// TIA Portal V17 export
// export: Created 2024-09-02T12:50:15.659418Z, ExportSetting WithDefaults, DisplayName Totally Integrated Automation Portal, DisplayVersion V17, DisplayName TIA Portal Openness, DisplayVersion V17, DisplayName TIA Portal Version Control Interface, DisplayVersion V17, DisplayName STEP 7 Professional, DisplayVersion V17, DisplayName STEP 7 Safety, DisplayVersion V17, DisplayName WinCC Professional, DisplayVersion V17
FUNCTION "AnwFC_ZP_InterfaceMainScreen_OP70" : Void   // FC163, LAD
TITLE = Station overview / Stationsübersicht
{ S7_Optimized_Access := 'TRUE' }
AUTHOR : OlegFuehrus
FAMILY : BA
NAME : BA
VERSION : 0.1
// stored: AutoNumber false, IsIECCheckEnabled false, SetENOAutomatically false, UDAEnableTagReadback false
   VAR_TEMP
      t_VKE0 : Bool;
      t_VKE1 : Bool;
   END_VAR
BEGIN

REGION Network 1: INIT
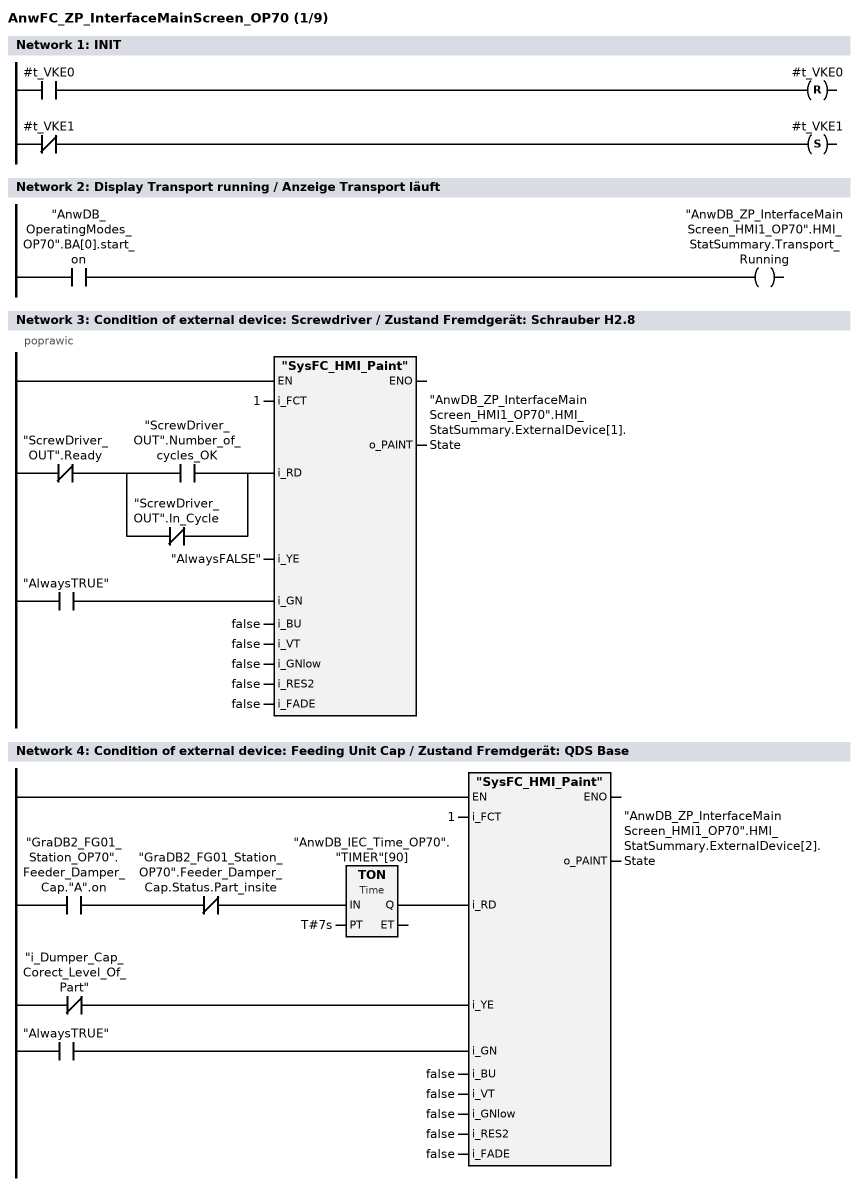
   RUNG wire#powerrail
      Contact( #t_VKE0 )
      R_Coil( #t_VKE0 )
   END_RUNG
   RUNG wire#powerrail
      I_Contact( #t_VKE1 )
      S_Coil( #t_VKE1 )
   END_RUNG
   // the same network as SCL:
   IF #t_VKE0 THEN #t_VKE0 := FALSE; END_IF;
   IF NOT #t_VKE1 THEN #t_VKE1 := TRUE; END_IF;
END_REGION

REGION Network 2: Display Transport running / Anzeige Transport läuft
   RUNG wire#powerrail
      Contact( "AnwDB_OperatingModes_OP70".BA[0].start_on )
      Coil( "AnwDB_ZP_InterfaceMainScreen_HMI1_OP70".HMI_StatSummary.Transport_Running )
   END_RUNG
   // the same network as SCL:
   "AnwDB_ZP_InterfaceMainScreen_HMI1_OP70".HMI_StatSummary.Transport_Running := "AnwDB_OperatingModes_OP70".BA[0].start_on;
END_REGION

REGION Network 3: Condition of external device: Screwdriver / Zustand Fremdgerät: Schrauber H2.8
   // poprawic
   RUNG wire#powerrail
      "SysFC_HMI_Paint"(i_RD := wire#w2, i_GN := wire#w3, i_FCT := 1, i_YE := "AlwaysFALSE", i_BU := false, i_VT := false, i_GNlow := false, i_RES2 := false, i_FADE := false, o_PAINT => "AnwDB_ZP_InterfaceMainScreen_HMI1_OP70".HMI_StatSummary.ExternalDevice[1].State)
   END_RUNG
   RUNG wire#powerrail
      I_Contact( "ScrewDriver_OUT".Ready )
      wire#w1
      Contact( "ScrewDriver_OUT".Number_of_cycles_OK )
   END_RUNG wire#w2
   RUNG wire#w1
      I_Contact( "ScrewDriver_OUT".In_Cycle )
   END_RUNG wire#w2
   RUNG wire#powerrail
      Contact( "AlwaysTRUE" )
   END_RUNG wire#w3
   // the same network as SCL:
   "SysFC_HMI_Paint"(i_FCT := 1,
                     i_RD := NOT "ScrewDriver_OUT".Ready AND ("ScrewDriver_OUT".Number_of_cycles_OK OR NOT "ScrewDriver_OUT".In_Cycle),
                     i_YE := "AlwaysFALSE",
                     i_GN := "AlwaysTRUE",
                     i_BU := false,
                     i_VT := false,
                     i_GNlow := false,
                     i_RES2 := false,
                     i_FADE := false,
                     o_PAINT => "AnwDB_ZP_InterfaceMainScreen_HMI1_OP70".HMI_StatSummary.ExternalDevice[1].State);
END_REGION

REGION Network 4: Condition of external device: Feeding Unit Cap / Zustand Fremdgerät: QDS Base
   RUNG wire#powerrail
      "SysFC_HMI_Paint"(i_RD := wire#w1, i_YE := wire#w2, i_GN := wire#w3, i_FCT := 1, i_BU := false, i_VT := false, i_GNlow := false, i_RES2 := false, i_FADE := false, o_PAINT => "AnwDB_ZP_InterfaceMainScreen_HMI1_OP70".HMI_StatSummary.ExternalDevice[2].State)
   END_RUNG
   RUNG wire#powerrail
      Contact( "GraDB2_FG01_Station_OP70".Feeder_Damper_Cap."A".on )
      I_Contact( "GraDB2_FG01_Station_OP70".Feeder_Damper_Cap.Status.Part_insite )
      { S7_Templates := "time_type := Time" } "AnwDB_IEC_Time_OP70"."TIMER"[90].TON(pt := T#7s, et =>)
   END_RUNG wire#w1
   RUNG wire#powerrail
      I_Contact( "i_Dumper_Cap_Corect_Level_Of_Part" )
   END_RUNG wire#w2
   RUNG wire#powerrail
      Contact( "AlwaysTRUE" )
   END_RUNG wire#w3
   // the same network as SCL:
   "AnwDB_IEC_Time_OP70"."TIMER"[90].TON(IN := "GraDB2_FG01_Station_OP70".Feeder_Damper_Cap."A".on AND NOT "GraDB2_FG01_Station_OP70".Feeder_Damper_Cap.Status.Part_insite,
                           PT := T#7s);
   "SysFC_HMI_Paint"(i_FCT := 1,
                     i_RD := "AnwDB_IEC_Time_OP70"."TIMER"[90].Q,
                     i_YE := NOT "i_Dumper_Cap_Corect_Level_Of_Part",
                     i_GN := "AlwaysTRUE",
                     i_BU := false,
                     i_VT := false,
                     i_GNlow := false,
                     i_RES2 := false,
                     i_FADE := false,
                     o_PAINT => "AnwDB_ZP_InterfaceMainScreen_HMI1_OP70".HMI_StatSummary.ExternalDevice[2].State);
END_REGION

REGION Network 5: Condition of external device: Feeding Unit Ball / Zustand Fremdgerät: Tox H2.10
   // dorobic
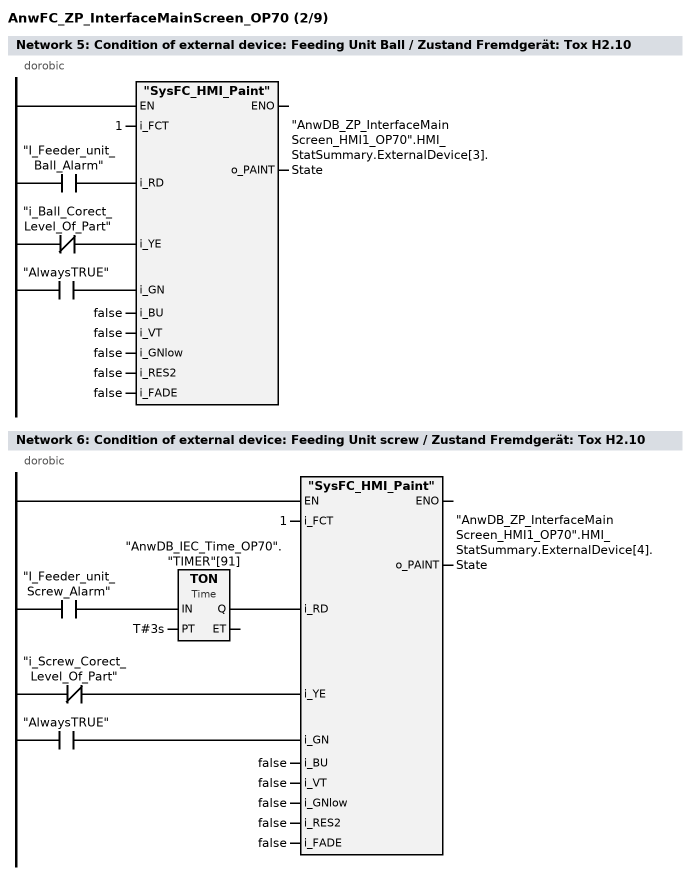
   RUNG wire#powerrail
      "SysFC_HMI_Paint"(i_RD := wire#w1, i_YE := wire#w2, i_GN := wire#w3, i_FCT := 1, i_BU := false, i_VT := false, i_GNlow := false, i_RES2 := false, i_FADE := false, o_PAINT => "AnwDB_ZP_InterfaceMainScreen_HMI1_OP70".HMI_StatSummary.ExternalDevice[3].State)
   END_RUNG
   RUNG wire#powerrail
      Contact( "I_Feeder_unit_Ball_Alarm" )
   END_RUNG wire#w1
   RUNG wire#powerrail
      I_Contact( "i_Ball_Corect_Level_Of_Part" )
   END_RUNG wire#w2
   RUNG wire#powerrail
      Contact( "AlwaysTRUE" )
   END_RUNG wire#w3
   // the same network as SCL:
   "SysFC_HMI_Paint"(i_FCT := 1,
                     i_RD := "I_Feeder_unit_Ball_Alarm",
                     i_YE := NOT "i_Ball_Corect_Level_Of_Part",
                     i_GN := "AlwaysTRUE",
                     i_BU := false,
                     i_VT := false,
                     i_GNlow := false,
                     i_RES2 := false,
                     i_FADE := false,
                     o_PAINT => "AnwDB_ZP_InterfaceMainScreen_HMI1_OP70".HMI_StatSummary.ExternalDevice[3].State);
END_REGION

REGION Network 6: Condition of external device: Feeding Unit screw / Zustand Fremdgerät: Tox H2.10
   // dorobic
   RUNG wire#powerrail
      "SysFC_HMI_Paint"(i_RD := wire#w1, i_YE := wire#w2, i_GN := wire#w3, i_FCT := 1, i_BU := false, i_VT := false, i_GNlow := false, i_RES2 := false, i_FADE := false, o_PAINT => "AnwDB_ZP_InterfaceMainScreen_HMI1_OP70".HMI_StatSummary.ExternalDevice[4].State)
   END_RUNG
   RUNG wire#powerrail
      Contact( "I_Feeder_unit_Screw_Alarm" )
      { S7_Templates := "time_type := Time" } "AnwDB_IEC_Time_OP70"."TIMER"[91].TON(pt := T#3s, et =>)
   END_RUNG wire#w1
   RUNG wire#powerrail
      I_Contact( "i_Screw_Corect_Level_Of_Part" )
   END_RUNG wire#w2
   RUNG wire#powerrail
      Contact( "AlwaysTRUE" )
   END_RUNG wire#w3
   // the same network as SCL:
   "AnwDB_IEC_Time_OP70"."TIMER"[91].TON(IN := "I_Feeder_unit_Screw_Alarm", PT := T#3s);
   "SysFC_HMI_Paint"(i_FCT := 1,
                     i_RD := "AnwDB_IEC_Time_OP70"."TIMER"[91].Q,
                     i_YE := NOT "i_Screw_Corect_Level_Of_Part",
                     i_GN := "AlwaysTRUE",
                     i_BU := false,
                     i_VT := false,
                     i_GNlow := false,
                     i_RES2 := false,
                     i_FADE := false,
                     o_PAINT => "AnwDB_ZP_InterfaceMainScreen_HMI1_OP70".HMI_StatSummary.ExternalDevice[4].State);
END_REGION

REGION Network 7: Condition of external device: Camera / Zustand Fremdgerät: Tox H2.10
   // dorobic
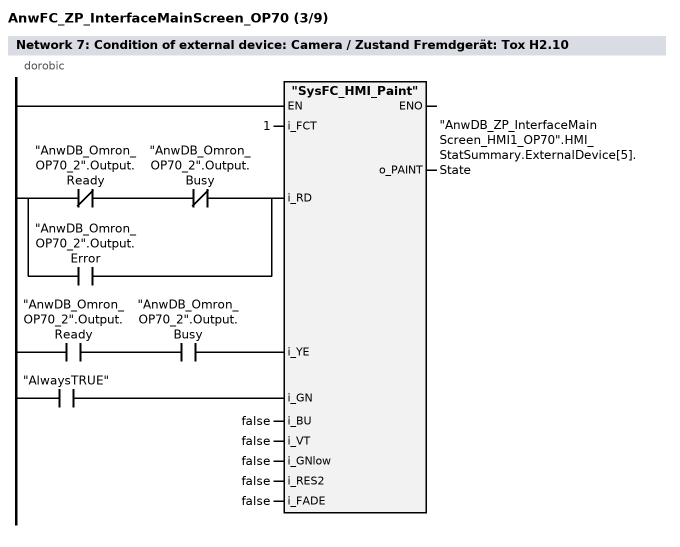
   RUNG wire#powerrail
      "SysFC_HMI_Paint"(i_RD := wire#w1, i_YE := wire#w2, i_GN := wire#w3, i_FCT := 1, i_BU := false, i_VT := false, i_GNlow := false, i_RES2 := false, i_FADE := false, o_PAINT => "AnwDB_ZP_InterfaceMainScreen_HMI1_OP70".HMI_StatSummary.ExternalDevice[5].State)
   END_RUNG
   RUNG wire#powerrail
      I_Contact( "AnwDB_Omron_OP70_2".Output.Ready )
      I_Contact( "AnwDB_Omron_OP70_2".Output.Busy )
   END_RUNG wire#w1
   RUNG wire#powerrail
      Contact( "AnwDB_Omron_OP70_2".Output.Error )
   END_RUNG wire#w1
   RUNG wire#powerrail
      Contact( "AnwDB_Omron_OP70_2".Output.Ready )
      Contact( "AnwDB_Omron_OP70_2".Output.Busy )
   END_RUNG wire#w2
   RUNG wire#powerrail
      Contact( "AlwaysTRUE" )
   END_RUNG wire#w3
   // the same network as SCL:
   "SysFC_HMI_Paint"(i_FCT := 1,
                     i_RD := (NOT "AnwDB_Omron_OP70_2".Output.Ready AND NOT "AnwDB_Omron_OP70_2".Output.Busy) OR "AnwDB_Omron_OP70_2".Output.Error,
                     i_YE := "AnwDB_Omron_OP70_2".Output.Ready AND "AnwDB_Omron_OP70_2".Output.Busy,
                     i_GN := "AlwaysTRUE",
                     i_BU := false,
                     i_VT := false,
                     i_GNlow := false,
                     i_RES2 := false,
                     i_FADE := false,
                     o_PAINT => "AnwDB_ZP_InterfaceMainScreen_HMI1_OP70".HMI_StatSummary.ExternalDevice[5].State);
END_REGION

REGION Network 8: Station overview [0] / Stationsübersicht [0]
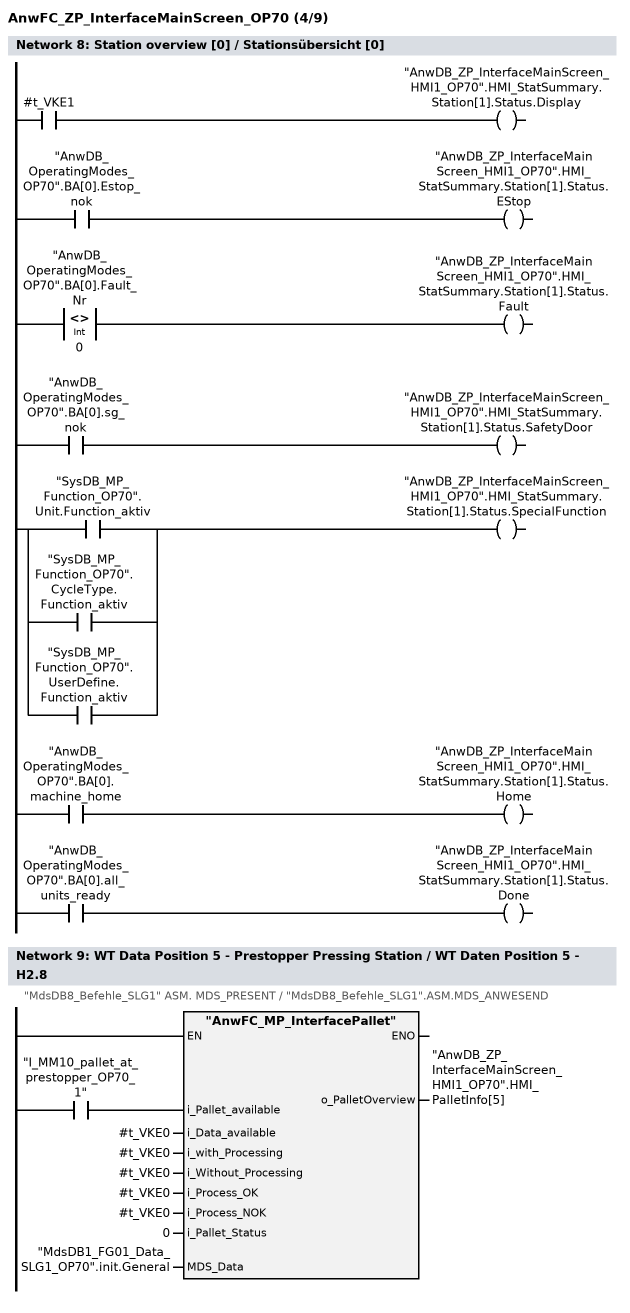
   RUNG wire#powerrail
      Contact( #t_VKE1 )
      Coil( "AnwDB_ZP_InterfaceMainScreen_HMI1_OP70".HMI_StatSummary.Station[1].Status.Display )
   END_RUNG
   RUNG wire#powerrail
      Contact( "AnwDB_OperatingModes_OP70".BA[0].Estop_nok )
      Coil( "AnwDB_ZP_InterfaceMainScreen_HMI1_OP70".HMI_StatSummary.Station[1].Status.EStop )
   END_RUNG
   RUNG wire#powerrail
      { S7_Templates := "SrcType := Int" } NE_Contact(in1 := "AnwDB_OperatingModes_OP70".BA[0].Fault_Nr, in2 := 0)
      Coil( "AnwDB_ZP_InterfaceMainScreen_HMI1_OP70".HMI_StatSummary.Station[1].Status.Fault )
   END_RUNG
   RUNG wire#powerrail
      Contact( "AnwDB_OperatingModes_OP70".BA[0].sg_nok )
      Coil( "AnwDB_ZP_InterfaceMainScreen_HMI1_OP70".HMI_StatSummary.Station[1].Status.SafetyDoor )
   END_RUNG
   RUNG wire#powerrail
      Contact( "SysDB_MP_Function_OP70".Unit.Function_aktiv )
      wire#w1
      Coil( "AnwDB_ZP_InterfaceMainScreen_HMI1_OP70".HMI_StatSummary.Station[1].Status.SpecialFunction )
   END_RUNG
   RUNG wire#powerrail
      Contact( "SysDB_MP_Function_OP70".CycleType.Function_aktiv )
   END_RUNG wire#w1
   RUNG wire#powerrail
      Contact( "SysDB_MP_Function_OP70".UserDefine.Function_aktiv )
   END_RUNG wire#w1
   RUNG wire#powerrail
      Contact( "AnwDB_OperatingModes_OP70".BA[0].machine_home )
      Coil( "AnwDB_ZP_InterfaceMainScreen_HMI1_OP70".HMI_StatSummary.Station[1].Status.Home )
   END_RUNG
   RUNG wire#powerrail
      Contact( "AnwDB_OperatingModes_OP70".BA[0].all_units_ready )
      Coil( "AnwDB_ZP_InterfaceMainScreen_HMI1_OP70".HMI_StatSummary.Station[1].Status.Done )
   END_RUNG
   // the same network as SCL:
   "AnwDB_ZP_InterfaceMainScreen_HMI1_OP70".HMI_StatSummary.Station[1].Status.Display := #t_VKE1;
   "AnwDB_ZP_InterfaceMainScreen_HMI1_OP70".HMI_StatSummary.Station[1].Status.EStop := "AnwDB_OperatingModes_OP70".BA[0].Estop_nok;
   "AnwDB_ZP_InterfaceMainScreen_HMI1_OP70".HMI_StatSummary.Station[1].Status.Fault := "AnwDB_OperatingModes_OP70".BA[0].Fault_Nr <> 0;
   "AnwDB_ZP_InterfaceMainScreen_HMI1_OP70".HMI_StatSummary.Station[1].Status.SafetyDoor := "AnwDB_OperatingModes_OP70".BA[0].sg_nok;
   "AnwDB_ZP_InterfaceMainScreen_HMI1_OP70".HMI_StatSummary.Station[1].Status.SpecialFunction := "SysDB_MP_Function_OP70".Unit.Function_aktiv OR "SysDB_MP_Function_OP70".CycleType.Function_aktiv OR "SysDB_MP_Function_OP70".UserDefine.Function_aktiv;
   "AnwDB_ZP_InterfaceMainScreen_HMI1_OP70".HMI_StatSummary.Station[1].Status.Home := "AnwDB_OperatingModes_OP70".BA[0].machine_home;
   "AnwDB_ZP_InterfaceMainScreen_HMI1_OP70".HMI_StatSummary.Station[1].Status.Done := "AnwDB_OperatingModes_OP70".BA[0].all_units_ready;
END_REGION

REGION Network 9: WT Data Position 5 - Prestopper Pressing Station / WT Daten Position 5 - H2.8
   // "MdsDB8_Befehle_SLG1" ASM. MDS_PRESENT / "MdsDB8_Befehle_SLG1".ASM.MDS_ANWESEND
   RUNG wire#powerrail
      "AnwFC_MP_InterfacePallet"(i_Pallet_available := wire#w1, i_Data_available := #t_VKE0, i_with_Processing := #t_VKE0, i_Without_Processing := #t_VKE0, i_Process_OK := #t_VKE0, i_Process_NOK := #t_VKE0, i_Pallet_Status := 0, MDS_Data := "MdsDB1_FG01_Data_SLG1_OP70".init.General, o_PalletOverview => "AnwDB_ZP_InterfaceMainScreen_HMI1_OP70".HMI_PalletInfo[5])
   END_RUNG
   RUNG wire#powerrail
      Contact( "I_MM10_pallet_at_prestopper_OP70_1" )
   END_RUNG wire#w1
   // the same network as SCL:
   "AnwFC_MP_InterfacePallet"(i_Pallet_available := "I_MM10_pallet_at_prestopper_OP70_1",
                           i_Data_available := #t_VKE0,
                           i_with_Processing := #t_VKE0,
                           i_Without_Processing := #t_VKE0,
                           i_Process_OK := #t_VKE0,
                           i_Process_NOK := #t_VKE0,
                           i_Pallet_Status := 0,
                           MDS_Data := "MdsDB1_FG01_Data_SLG1_OP70".init.General,
                           o_PalletOverview => "AnwDB_ZP_InterfaceMainScreen_HMI1_OP70".HMI_PalletInfo[5]);
END_REGION

REGION Network 10: WT Data Position 4 - Stopper Pressing Station / WT Daten Position 4 - H2.9
   // "MdsDB8_Befehle_SLG1" ASM. MDS_PRESENT / "MdsDB8_Befehle_SLG1".ASM.MDS_ANWESEND
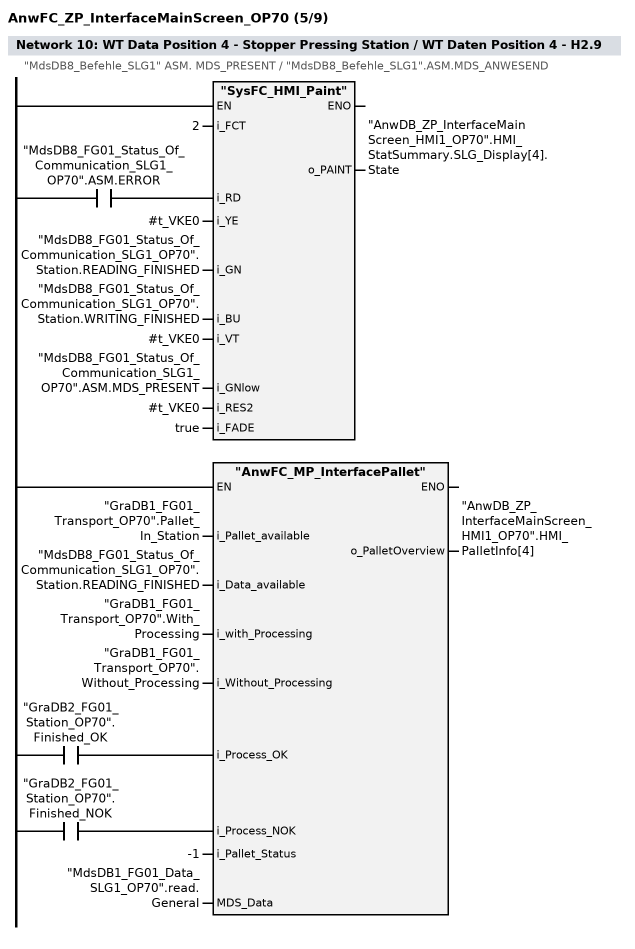
   RUNG wire#powerrail
      "SysFC_HMI_Paint"(i_RD := wire#w1, i_FCT := 2, i_YE := #t_VKE0, i_GN := "MdsDB8_FG01_Status_Of_Communication_SLG1_OP70".Station.READING_FINISHED, i_BU := "MdsDB8_FG01_Status_Of_Communication_SLG1_OP70".Station.WRITING_FINISHED, i_VT := #t_VKE0, i_GNlow := "MdsDB8_FG01_Status_Of_Communication_SLG1_OP70".ASM.MDS_PRESENT, i_RES2 := #t_VKE0, i_FADE := true, o_PAINT => "AnwDB_ZP_InterfaceMainScreen_HMI1_OP70".HMI_StatSummary.SLG_Display[4].State)
   END_RUNG
   RUNG wire#powerrail
      Contact( "MdsDB8_FG01_Status_Of_Communication_SLG1_OP70".ASM.ERROR )
   END_RUNG wire#w1
   RUNG wire#powerrail
      "AnwFC_MP_InterfacePallet"(i_Process_OK := wire#w2, i_Process_NOK := wire#w3, i_Pallet_available := "GraDB1_FG01_Transport_OP70".Pallet_In_Station, i_Data_available := "MdsDB8_FG01_Status_Of_Communication_SLG1_OP70".Station.READING_FINISHED, i_with_Processing := "GraDB1_FG01_Transport_OP70".With_Processing, i_Without_Processing := "GraDB1_FG01_Transport_OP70".Without_Processing, i_Pallet_Status := -1, MDS_Data := "MdsDB1_FG01_Data_SLG1_OP70".read.General, o_PalletOverview => "AnwDB_ZP_InterfaceMainScreen_HMI1_OP70".HMI_PalletInfo[4])
   END_RUNG
   RUNG wire#powerrail
      Contact( "GraDB2_FG01_Station_OP70".Finished_OK )
   END_RUNG wire#w2
   RUNG wire#powerrail
      Contact( "GraDB2_FG01_Station_OP70".Finished_NOK )
   END_RUNG wire#w3
   // the same network as SCL:
   "SysFC_HMI_Paint"(i_FCT := 2,
                     i_RD := "MdsDB8_FG01_Status_Of_Communication_SLG1_OP70".ASM.ERROR,
                     i_YE := #t_VKE0,
                     i_GN := "MdsDB8_FG01_Status_Of_Communication_SLG1_OP70".Station.READING_FINISHED,
                     i_BU := "MdsDB8_FG01_Status_Of_Communication_SLG1_OP70".Station.WRITING_FINISHED,
                     i_VT := #t_VKE0,
                     i_GNlow := "MdsDB8_FG01_Status_Of_Communication_SLG1_OP70".ASM.MDS_PRESENT,
                     i_RES2 := #t_VKE0,
                     i_FADE := true,
                     o_PAINT => "AnwDB_ZP_InterfaceMainScreen_HMI1_OP70".HMI_StatSummary.SLG_Display[4].State);
   "AnwFC_MP_InterfacePallet"(i_Pallet_available := "GraDB1_FG01_Transport_OP70".Pallet_In_Station,
                           i_Data_available := "MdsDB8_FG01_Status_Of_Communication_SLG1_OP70".Station.READING_FINISHED,
                           i_with_Processing := "GraDB1_FG01_Transport_OP70".With_Processing,
                           i_Without_Processing := "GraDB1_FG01_Transport_OP70".Without_Processing,
                           i_Process_OK := "GraDB2_FG01_Station_OP70".Finished_OK,
                           i_Process_NOK := "GraDB2_FG01_Station_OP70".Finished_NOK,
                           i_Pallet_Status := -1,
                           MDS_Data := "MdsDB1_FG01_Data_SLG1_OP70".read.General,
                           o_PalletOverview => "AnwDB_ZP_InterfaceMainScreen_HMI1_OP70".HMI_PalletInfo[4]);
END_REGION

REGION Network 11: WT Data Position 3 - Prestopper Camera Station / WT Daten Position 3 - H2.10
   // "MdsDB8_Befehle_SLG3" ASM. MDS_PRESENT / "MdsDB8_Befehle_slg3".ASM.MDS_ANWESEND
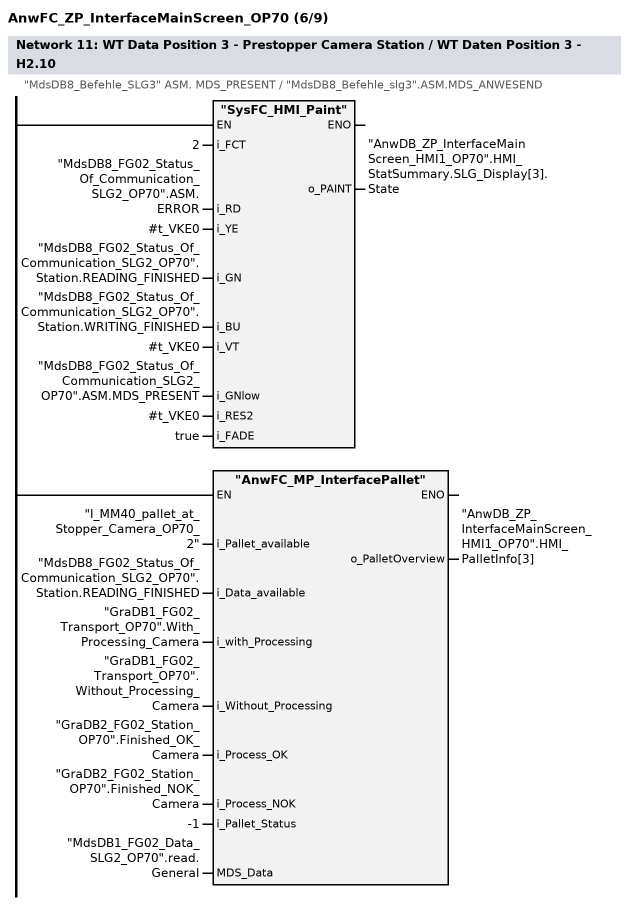
   RUNG wire#powerrail
      "SysFC_HMI_Paint"(i_FCT := 2, i_RD := "MdsDB8_FG02_Status_Of_Communication_SLG2_OP70".ASM.ERROR, i_YE := #t_VKE0, i_GN := "MdsDB8_FG02_Status_Of_Communication_SLG2_OP70".Station.READING_FINISHED, i_BU := "MdsDB8_FG02_Status_Of_Communication_SLG2_OP70".Station.WRITING_FINISHED, i_VT := #t_VKE0, i_GNlow := "MdsDB8_FG02_Status_Of_Communication_SLG2_OP70".ASM.MDS_PRESENT, i_RES2 := #t_VKE0, i_FADE := true, o_PAINT => "AnwDB_ZP_InterfaceMainScreen_HMI1_OP70".HMI_StatSummary.SLG_Display[3].State)
   END_RUNG
   RUNG wire#powerrail
      "AnwFC_MP_InterfacePallet"(i_Pallet_available := "I_MM40_pallet_at_Stopper_Camera_OP70_2", i_Data_available := "MdsDB8_FG02_Status_Of_Communication_SLG2_OP70".Station.READING_FINISHED, i_with_Processing := "GraDB1_FG02_Transport_OP70".With_Processing_Camera, i_Without_Processing := "GraDB1_FG02_Transport_OP70".Without_Processing_Camera, i_Process_OK := "GraDB2_FG02_Station_OP70".Finished_OK_Camera, i_Process_NOK := "GraDB2_FG02_Station_OP70".Finished_NOK_Camera, i_Pallet_Status := -1, MDS_Data := "MdsDB1_FG02_Data_SLG2_OP70".read.General, o_PalletOverview => "AnwDB_ZP_InterfaceMainScreen_HMI1_OP70".HMI_PalletInfo[3])
   END_RUNG
   // the same network as SCL:
   "SysFC_HMI_Paint"(i_FCT := 2,
                     i_RD := "MdsDB8_FG02_Status_Of_Communication_SLG2_OP70".ASM.ERROR,
                     i_YE := #t_VKE0,
                     i_GN := "MdsDB8_FG02_Status_Of_Communication_SLG2_OP70".Station.READING_FINISHED,
                     i_BU := "MdsDB8_FG02_Status_Of_Communication_SLG2_OP70".Station.WRITING_FINISHED,
                     i_VT := #t_VKE0,
                     i_GNlow := "MdsDB8_FG02_Status_Of_Communication_SLG2_OP70".ASM.MDS_PRESENT,
                     i_RES2 := #t_VKE0,
                     i_FADE := true,
                     o_PAINT => "AnwDB_ZP_InterfaceMainScreen_HMI1_OP70".HMI_StatSummary.SLG_Display[3].State);
   "AnwFC_MP_InterfacePallet"(i_Pallet_available := "I_MM40_pallet_at_Stopper_Camera_OP70_2",
                           i_Data_available := "MdsDB8_FG02_Status_Of_Communication_SLG2_OP70".Station.READING_FINISHED,
                           i_with_Processing := "GraDB1_FG02_Transport_OP70".With_Processing_Camera,
                           i_Without_Processing := "GraDB1_FG02_Transport_OP70".Without_Processing_Camera,
                           i_Process_OK := "GraDB2_FG02_Station_OP70".Finished_OK_Camera,
                           i_Process_NOK := "GraDB2_FG02_Station_OP70".Finished_NOK_Camera,
                           i_Pallet_Status := -1,
                           MDS_Data := "MdsDB1_FG02_Data_SLG2_OP70".read.General,
                           o_PalletOverview => "AnwDB_ZP_InterfaceMainScreen_HMI1_OP70".HMI_PalletInfo[3]);
END_REGION

REGION Network 12: WT Data Position 2 - Stopper Screwdriver Station / WT Daten Position 3 - H2.10
   // "MdsDB8_Befehle_SLG3" ASM. MDS_PRESENT / "MdsDB8_Befehle_slg3".ASM.MDS_ANWESEND
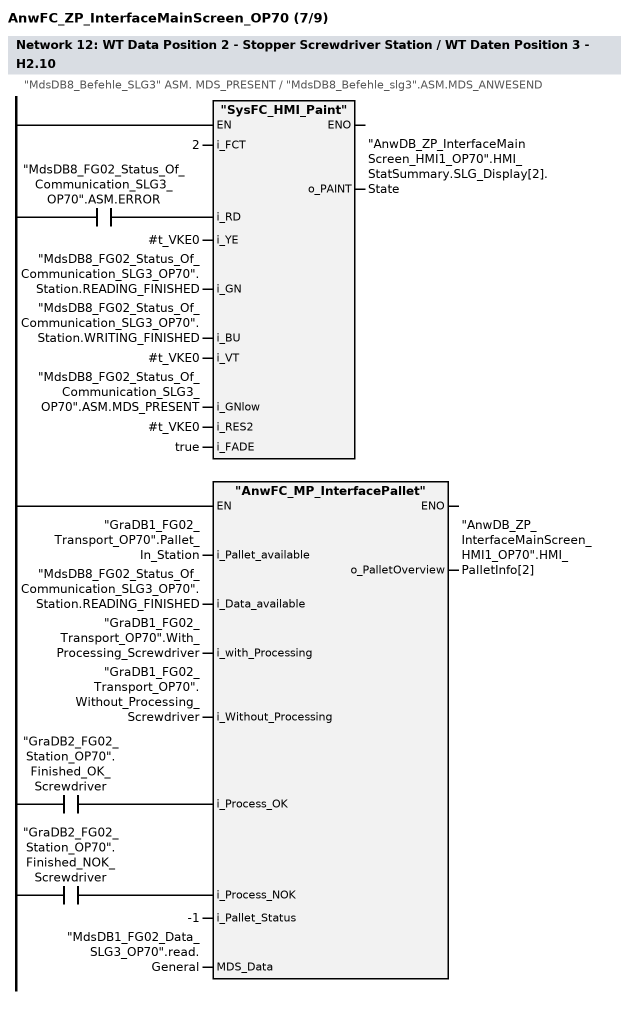
   RUNG wire#powerrail
      "SysFC_HMI_Paint"(i_RD := wire#w1, i_FCT := 2, i_YE := #t_VKE0, i_GN := "MdsDB8_FG02_Status_Of_Communication_SLG3_OP70".Station.READING_FINISHED, i_BU := "MdsDB8_FG02_Status_Of_Communication_SLG3_OP70".Station.WRITING_FINISHED, i_VT := #t_VKE0, i_GNlow := "MdsDB8_FG02_Status_Of_Communication_SLG3_OP70".ASM.MDS_PRESENT, i_RES2 := #t_VKE0, i_FADE := true, o_PAINT => "AnwDB_ZP_InterfaceMainScreen_HMI1_OP70".HMI_StatSummary.SLG_Display[2].State)
   END_RUNG
   RUNG wire#powerrail
      Contact( "MdsDB8_FG02_Status_Of_Communication_SLG3_OP70".ASM.ERROR )
   END_RUNG wire#w1
   RUNG wire#powerrail
      "AnwFC_MP_InterfacePallet"(i_Process_OK := wire#w2, i_Process_NOK := wire#w3, i_Pallet_available := "GraDB1_FG02_Transport_OP70".Pallet_In_Station, i_Data_available := "MdsDB8_FG02_Status_Of_Communication_SLG3_OP70".Station.READING_FINISHED, i_with_Processing := "GraDB1_FG02_Transport_OP70".With_Processing_Screwdriver, i_Without_Processing := "GraDB1_FG02_Transport_OP70".Without_Processing_Screwdriver, i_Pallet_Status := -1, MDS_Data := "MdsDB1_FG02_Data_SLG3_OP70".read.General, o_PalletOverview => "AnwDB_ZP_InterfaceMainScreen_HMI1_OP70".HMI_PalletInfo[2])
   END_RUNG
   RUNG wire#powerrail
      Contact( "GraDB2_FG02_Station_OP70".Finished_OK_Screwdriver )
   END_RUNG wire#w2
   RUNG wire#powerrail
      Contact( "GraDB2_FG02_Station_OP70".Finished_NOK_Screwdriver )
   END_RUNG wire#w3
   // the same network as SCL:
   "SysFC_HMI_Paint"(i_FCT := 2,
                     i_RD := "MdsDB8_FG02_Status_Of_Communication_SLG3_OP70".ASM.ERROR,
                     i_YE := #t_VKE0,
                     i_GN := "MdsDB8_FG02_Status_Of_Communication_SLG3_OP70".Station.READING_FINISHED,
                     i_BU := "MdsDB8_FG02_Status_Of_Communication_SLG3_OP70".Station.WRITING_FINISHED,
                     i_VT := #t_VKE0,
                     i_GNlow := "MdsDB8_FG02_Status_Of_Communication_SLG3_OP70".ASM.MDS_PRESENT,
                     i_RES2 := #t_VKE0,
                     i_FADE := true,
                     o_PAINT => "AnwDB_ZP_InterfaceMainScreen_HMI1_OP70".HMI_StatSummary.SLG_Display[2].State);
   "AnwFC_MP_InterfacePallet"(i_Pallet_available := "GraDB1_FG02_Transport_OP70".Pallet_In_Station,
                           i_Data_available := "MdsDB8_FG02_Status_Of_Communication_SLG3_OP70".Station.READING_FINISHED,
                           i_with_Processing := "GraDB1_FG02_Transport_OP70".With_Processing_Screwdriver,
                           i_Without_Processing := "GraDB1_FG02_Transport_OP70".Without_Processing_Screwdriver,
                           i_Process_OK := "GraDB2_FG02_Station_OP70".Finished_OK_Screwdriver,
                           i_Process_NOK := "GraDB2_FG02_Station_OP70".Finished_NOK_Screwdriver,
                           i_Pallet_Status := -1,
                           MDS_Data := "MdsDB1_FG02_Data_SLG3_OP70".read.General,
                           o_PalletOverview => "AnwDB_ZP_InterfaceMainScreen_HMI1_OP70".HMI_PalletInfo[2]);
END_REGION

REGION Network 13: Wrie pallet status On the main screen 70.1
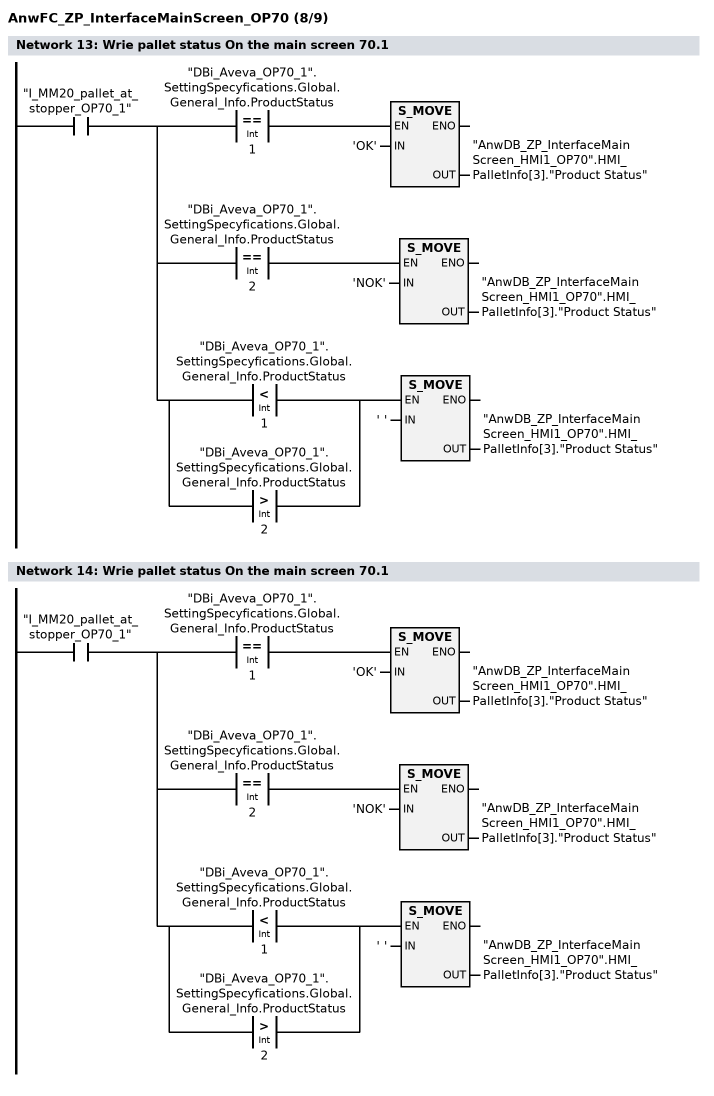
   RUNG wire#powerrail
      Contact( "I_MM20_pallet_at_stopper_OP70_1" )
      wire#w1
      { S7_Templates := "SrcType := Int" } EQ_Contact(in1 := "DBi_Aveva_OP70_1".SettingSpecyfications.Global.General_Info.ProductStatus, in2 := 1)
      S_Move(in := 'OK', out => "AnwDB_ZP_InterfaceMainScreen_HMI1_OP70".HMI_PalletInfo[3]."Product Status")
   END_RUNG
   RUNG wire#w1
      { S7_Templates := "SrcType := Int" } EQ_Contact(in1 := "DBi_Aveva_OP70_1".SettingSpecyfications.Global.General_Info.ProductStatus, in2 := 2)
      S_Move(in := 'NOK', out => "AnwDB_ZP_InterfaceMainScreen_HMI1_OP70".HMI_PalletInfo[3]."Product Status")
   END_RUNG
   RUNG wire#w1
      { S7_Templates := "SrcType := Int" } LT_Contact(in1 := "DBi_Aveva_OP70_1".SettingSpecyfications.Global.General_Info.ProductStatus, in2 := 1)
      wire#w2
      S_Move(in := ' ', out => "AnwDB_ZP_InterfaceMainScreen_HMI1_OP70".HMI_PalletInfo[3]."Product Status")
   END_RUNG
   RUNG wire#w1
      { S7_Templates := "SrcType := Int" } GT_Contact(in1 := "DBi_Aveva_OP70_1".SettingSpecyfications.Global.General_Info.ProductStatus, in2 := 2)
   END_RUNG wire#w2
   // the same network as SCL:
   IF "I_MM20_pallet_at_stopper_OP70_1" AND ("DBi_Aveva_OP70_1".SettingSpecyfications.Global.General_Info.ProductStatus = 1) THEN
       "AnwDB_ZP_InterfaceMainScreen_HMI1_OP70".HMI_PalletInfo[3]."Product Status" := 'OK';
   END_IF;
   IF "I_MM20_pallet_at_stopper_OP70_1" AND ("DBi_Aveva_OP70_1".SettingSpecyfications.Global.General_Info.ProductStatus = 2) THEN
       "AnwDB_ZP_InterfaceMainScreen_HMI1_OP70".HMI_PalletInfo[3]."Product Status" := 'NOK';
   END_IF;
   IF "I_MM20_pallet_at_stopper_OP70_1" AND (("DBi_Aveva_OP70_1".SettingSpecyfications.Global.General_Info.ProductStatus < 1) OR ("DBi_Aveva_OP70_1".SettingSpecyfications.Global.General_Info.ProductStatus > 2)) THEN
       "AnwDB_ZP_InterfaceMainScreen_HMI1_OP70".HMI_PalletInfo[3]."Product Status" := ' ';
   END_IF;
END_REGION

REGION Network 14: Wrie pallet status On the main screen 70.1
   RUNG wire#powerrail
      Contact( "I_MM20_pallet_at_stopper_OP70_1" )
      wire#w1
      { S7_Templates := "SrcType := Int" } EQ_Contact(in1 := "DBi_Aveva_OP70_1".SettingSpecyfications.Global.General_Info.ProductStatus, in2 := 1)
      S_Move(in := 'OK', out => "AnwDB_ZP_InterfaceMainScreen_HMI1_OP70".HMI_PalletInfo[3]."Product Status")
   END_RUNG
   RUNG wire#w1
      { S7_Templates := "SrcType := Int" } EQ_Contact(in1 := "DBi_Aveva_OP70_1".SettingSpecyfications.Global.General_Info.ProductStatus, in2 := 2)
      S_Move(in := 'NOK', out => "AnwDB_ZP_InterfaceMainScreen_HMI1_OP70".HMI_PalletInfo[3]."Product Status")
   END_RUNG
   RUNG wire#w1
      { S7_Templates := "SrcType := Int" } LT_Contact(in1 := "DBi_Aveva_OP70_1".SettingSpecyfications.Global.General_Info.ProductStatus, in2 := 1)
      wire#w2
      S_Move(in := ' ', out => "AnwDB_ZP_InterfaceMainScreen_HMI1_OP70".HMI_PalletInfo[3]."Product Status")
   END_RUNG
   RUNG wire#w1
      { S7_Templates := "SrcType := Int" } GT_Contact(in1 := "DBi_Aveva_OP70_1".SettingSpecyfications.Global.General_Info.ProductStatus, in2 := 2)
   END_RUNG wire#w2
   // the same network as SCL:
   IF "I_MM20_pallet_at_stopper_OP70_1" AND ("DBi_Aveva_OP70_1".SettingSpecyfications.Global.General_Info.ProductStatus = 1) THEN
       "AnwDB_ZP_InterfaceMainScreen_HMI1_OP70".HMI_PalletInfo[3]."Product Status" := 'OK';
   END_IF;
   IF "I_MM20_pallet_at_stopper_OP70_1" AND ("DBi_Aveva_OP70_1".SettingSpecyfications.Global.General_Info.ProductStatus = 2) THEN
       "AnwDB_ZP_InterfaceMainScreen_HMI1_OP70".HMI_PalletInfo[3]."Product Status" := 'NOK';
   END_IF;
   IF "I_MM20_pallet_at_stopper_OP70_1" AND (("DBi_Aveva_OP70_1".SettingSpecyfications.Global.General_Info.ProductStatus < 1) OR ("DBi_Aveva_OP70_1".SettingSpecyfications.Global.General_Info.ProductStatus > 2)) THEN
       "AnwDB_ZP_InterfaceMainScreen_HMI1_OP70".HMI_PalletInfo[3]."Product Status" := ' ';
   END_IF;
END_REGION

REGION Network 15: Wrie pallet status On the main screen 70.1
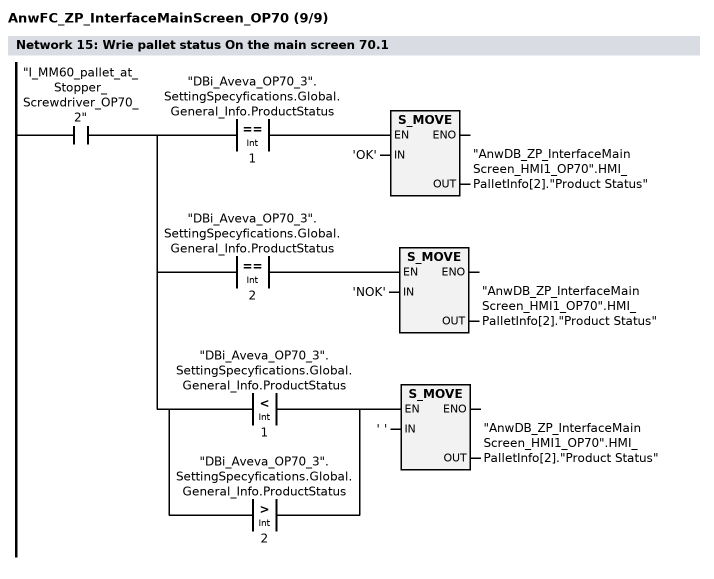
   RUNG wire#powerrail
      Contact( "I_MM60_pallet_at_Stopper_Screwdriver_OP70_2" )
      wire#w1
      { S7_Templates := "SrcType := Int" } EQ_Contact(in1 := "DBi_Aveva_OP70_3".SettingSpecyfications.Global.General_Info.ProductStatus, in2 := 1)
      S_Move(in := 'OK', out => "AnwDB_ZP_InterfaceMainScreen_HMI1_OP70".HMI_PalletInfo[2]."Product Status")
   END_RUNG
   RUNG wire#w1
      { S7_Templates := "SrcType := Int" } EQ_Contact(in1 := "DBi_Aveva_OP70_3".SettingSpecyfications.Global.General_Info.ProductStatus, in2 := 2)
      S_Move(in := 'NOK', out => "AnwDB_ZP_InterfaceMainScreen_HMI1_OP70".HMI_PalletInfo[2]."Product Status")
   END_RUNG
   RUNG wire#w1
      { S7_Templates := "SrcType := Int" } LT_Contact(in1 := "DBi_Aveva_OP70_3".SettingSpecyfications.Global.General_Info.ProductStatus, in2 := 1)
      wire#w2
      S_Move(in := ' ', out => "AnwDB_ZP_InterfaceMainScreen_HMI1_OP70".HMI_PalletInfo[2]."Product Status")
   END_RUNG
   RUNG wire#w1
      { S7_Templates := "SrcType := Int" } GT_Contact(in1 := "DBi_Aveva_OP70_3".SettingSpecyfications.Global.General_Info.ProductStatus, in2 := 2)
   END_RUNG wire#w2
   // the same network as SCL:
   IF "I_MM60_pallet_at_Stopper_Screwdriver_OP70_2" AND ("DBi_Aveva_OP70_3".SettingSpecyfications.Global.General_Info.ProductStatus = 1) THEN
       "AnwDB_ZP_InterfaceMainScreen_HMI1_OP70".HMI_PalletInfo[2]."Product Status" := 'OK';
   END_IF;
   IF "I_MM60_pallet_at_Stopper_Screwdriver_OP70_2" AND ("DBi_Aveva_OP70_3".SettingSpecyfications.Global.General_Info.ProductStatus = 2) THEN
       "AnwDB_ZP_InterfaceMainScreen_HMI1_OP70".HMI_PalletInfo[2]."Product Status" := 'NOK';
   END_IF;
   IF "I_MM60_pallet_at_Stopper_Screwdriver_OP70_2" AND (("DBi_Aveva_OP70_3".SettingSpecyfications.Global.General_Info.ProductStatus < 1) OR ("DBi_Aveva_OP70_3".SettingSpecyfications.Global.General_Info.ProductStatus > 2)) THEN
       "AnwDB_ZP_InterfaceMainScreen_HMI1_OP70".HMI_PalletInfo[2]."Product Status" := ' ';
   END_IF;
END_REGION
END_FUNCTION
